TYPE DMX_Status :
STRUCT
	TransmitAccepted : BIT;
	RecieveToggle : BIT;
	CyclicTxD_Disabled : BIT;
	DefaultDataSent : BIT;
	FrameSentToggle : BIT;
	TxPdoToggle : BIT;
	ChannelLength : UINT;
	StartCode : USINT;
END_STRUCT
END_TYPE

(* stored: Version 1.1.0.1
   DUT DMX_Status: Id {4f497bbd-1451-443c-9515-30040aba4375} *)
